Universal Robots PolyScope program: Put_into_box_E-series_UR3.urp

Program  (createdIn=3.0.0.0 lastSavedIn=5.0.3.30563)
Robot Program (runOnlyOnce=true speed=0 acceleration=0 useActiveTCP=false positionType=CartesianPose) feature=Base
  Set NoAction (payload=0 tcpAsCog=true)
  MoveJ speed 50 deg/s, acceleration 100 deg/s^2 (useActiveTCP=false positionType=JointAngles)
    Waypoint Home: TCP in base x=-0.556 y=-222.914 z=694.011 mm, rx=0.002 ry=-2.2182 rz=2.2173 rad; joints [0, -90.004, 0, -90.005, 0, 0] deg
    Waypoint End: TCP in base x=-222.255 y=-140.418 z=254.023 mm, rx=1.2057 ry=-1.2004 rz=-1.2169 rad; joints [-90, -180, 152, -242, 0, 270] deg
